{attribute 'qualified_only'}
//{attribute 'strict'}
TYPE eSMSStatus :
(
	Idle 			:= 	0,
	NewMessage 		:= 	1,
	SendingMessage 	:= 	2,
	error			:=	3
);
END_TYPE

(* stored: Version 1.1.0.1, ProductVersion 3.1.4026.18
   DUT eSMSStatus: Id {dfe4baa2-966c-45f1-aa3a-1690953db6ec} *)
